PROGRAM PRG_TEST
VAR
	_test : FB_Cylinder_Test;
END_VAR

TcUnit.RUN();

END_PROGRAM

(* stored: Version 1.1.0.1, ProductVersion 3.1.4026.17
   POU PRG_TEST: Id {58c96f65-a512-401a-b154-ddc116720dca}, SpecialFunc None *)
